// TIA Portal V17 export
// export: Created 2026-04-13T11:12:52.670393Z, ExportSetting WithDefaults, DisplayName Totally Integrated Automation Portal, DisplayVersion V17 Update 4, DisplayName TIA Portal Openness, DisplayVersion V17 Update 4, DisplayName TIA Portal Version Control Interface, DisplayVersion V17, DisplayName SINAMICS Startdrive Advanced, DisplayVersion V17, DisplayName SINAMICS Startdrive G130, G150, S120, S150, SINAMICS MV, S210, DisplayVersion V17, DisplayName SINAMICS Startdrive G110M, G120, G120C, G120D, G120P, G115D, DisplayVersion V17, DisplayName STEP 7 Professional, DisplayVersion V17 Update 4, DisplayName STEP 7 Safety, DisplayVersion V17, DisplayName WinCC Professional, DisplayVersion V17 Update 4
TagTable "OUTCIPJS"
  OUTCIPJS_1设定时间 : Real  (PLC tag OUTCIPJS.1设定时间, HMI_连接_1, 1 s)
  OUTCIPJS_2设定时间 : Real  (PLC tag OUTCIPJS.2设定时间, HMI_连接_1, 1 s)
  OUTCIPJS_3设定时间 : Real  (PLC tag OUTCIPJS.3设定时间, HMI_连接_1, 1 s)
  OUTCIPJS_4设定时间 : Real  (PLC tag OUTCIPJS.4设定时间, HMI_连接_1, 1 s)
  OUTCIPJS_5设定时间 : Real  (PLC tag OUTCIPJS.5设定时间, HMI_连接_1, 1 s)
  OUTCIPJS_6设定时间 : Real  (PLC tag OUTCIPJS.6设定时间, HMI_连接_1, 1 s)
  OUTCIPJS_7设定时间 : Real  (PLC tag OUTCIPJS.7设定时间, HMI_连接_1, 1 s)
  OUTCIPJS_8设定时间 : Real  (PLC tag OUTCIPJS.8设定时间, HMI_连接_1, 1 s)
  OUTCIPJS_9设定时间 : Real  (PLC tag OUTCIPJS.9设定时间, HMI_连接_1, 1 s)
  OUTCIPJS_10设定时间 : Real  (PLC tag OUTCIPJS.10设定时间, HMI_连接_1, 1 s)
  OUTCIPJS_11设定时间 : Real  (PLC tag OUTCIPJS.11设定时间, HMI_连接_1, 1 s)
  OUTCIPJS_12设定时间 : Real  (PLC tag OUTCIPJS.12设定时间, HMI_连接_1, 1 s)
  OUTCIPJS_13设定时间 : Real  (PLC tag OUTCIPJS.13设定时间, HMI_连接_1, 1 s)
  OUTCIPJS_14设定时间 : Real  (PLC tag OUTCIPJS.14设定时间, HMI_连接_1, 1 s)
  OUTCIPJS_15设定时间 : Real  (PLC tag OUTCIPJS.15设定时间, HMI_连接_1, 1 s)
  OUTCIPJS_16设定时间 : Real  (PLC tag OUTCIPJS.16设定时间, HMI_连接_1, 1 s)
  OUTCIPJS_1计时 : Real  (PLC tag OUTCIPJS.1计时, HMI_连接_1, 1 s)
  OUTCIPJS_2计时 : Real  (PLC tag OUTCIPJS.2计时, HMI_连接_1, 1 s)
  OUTCIPJS_3计时 : Real  (PLC tag OUTCIPJS.3计时, HMI_连接_1, 1 s)
  OUTCIPJS_4计时 : Real  (PLC tag OUTCIPJS.4计时, HMI_连接_1, 1 s)
  OUTCIPJS_5计时 : Real  (PLC tag OUTCIPJS.5计时, HMI_连接_1, 1 s)
  OUTCIPJS_6计时 : Real  (PLC tag OUTCIPJS.6计时, HMI_连接_1, 1 s)
  OUTCIPJS_7计时 : Real  (PLC tag OUTCIPJS.7计时, HMI_连接_1, 1 s)
  OUTCIPJS_8计时 : Real  (PLC tag OUTCIPJS.8计时, HMI_连接_1, 1 s)
  OUTCIPJS_9计时 : Real  (PLC tag OUTCIPJS.9计时, HMI_连接_1, 1 s)
  OUTCIPJS_10计时 : Real  (PLC tag OUTCIPJS.10计时, HMI_连接_1, 1 s)
  OUTCIPJS_11计时 : Real  (PLC tag OUTCIPJS.11计时, HMI_连接_1, 1 s)
  OUTCIPJS_12计时 : Real  (PLC tag OUTCIPJS.12计时, HMI_连接_1, 1 s)
  OUTCIPJS_13计时 : Real  (PLC tag OUTCIPJS.13计时, HMI_连接_1, 1 s)
  OUTCIPJS_14计时 : Real  (PLC tag OUTCIPJS.14计时, HMI_连接_1, 1 s)
  OUTCIPJS_15计时 : Real  (PLC tag OUTCIPJS.15计时, HMI_连接_1, 1 s)
  OUTCIPJS_16计时 : Real  (PLC tag OUTCIPJS.16计时, HMI_连接_1, 1 s)
